PROGRAM MAIN
VAR
END_VAR

END_PROGRAM

(* stored: Version 1.1.0.1
   POU MAIN: Id {27e010f8-6586-4164-9eaa-8d2a7e6065ce} *)
